TYPE ST_FireDetectionGet :
STRUCT
	SmokeDetected		:	BOOL;					//-1 if inoperative.
	CODetectorValues 	:  	ARRAY[0..2] OF REAL;	//-1 if inoperative.
	
	Events	:	ST_FireSystem_Events;
END_STRUCT
END_TYPE

(* stored: Version 1.1.0.1, ProductVersion 3.1.4024.12
   DUT ST_FireDetectionGet: Id {6cc78167-32bf-4519-8037-010d2b675e1a} *)
